KUKA KRL program: Bolge_1_Palet_Ort.src, Bolge_1_Palet_Ort.dat

--- Bolge_1_Palet_Ort.src ---
&ACCESS RVO1
&REL 27
&PARAM EDITMASK = *
&PARAM TEMPLATE = C:\KRC\Roboter\Template\vorgabe
&PARAM DISKPATH = KRC:\R1\Program\Sub_Rutinler
DEF Bolge_1_Palet_Ort( )
;FOLD INI;%{PE}
  ;FOLD BASISTECH INI
    GLOBAL INTERRUPT DECL 3 WHEN $STOPMESS==TRUE DO IR_STOPM ( )
    INTERRUPT ON 3
    BAS (#INITMOV,0 )
  ;ENDFOLD (BASISTECH INI)
  ;FOLD USER INI
    ;Make your modifications here

  ;ENDFOLD (USER INI)
;ENDFOLD (INI)

;;FOLD SPTP B1_Master Vel=100 % PDAT1 Tool[1]:Gripper Base[0] ;%{PE}
;;FOLD Parameters ;%{h}
;;Params IlfProvider=kukaroboter.basistech.inlineforms.movement.spline; Kuka.IsGlobalPoint=False; Kuka.PointName=B1_Master; Kuka.BlendingEnabled=False; Kuka.MoveDataPtpName=PDAT1; Kuka.VelocityPtp=100; Kuka.VelocityFieldEnabled=True; Kuka.ColDetectFieldEnabled=True; Kuka.CurrentCDSetIndex=0; Kuka.MovementParameterFieldEnabled=True; IlfCommand=SPTP
;;ENDFOLD
;SPTP XB1_Master WITH $VEL_AXIS[1] = SVEL_JOINT(100.0), $TOOL = STOOL2(FB1_Master), $BASE = SBASE(FB1_Master.BASE_NO), $IPO_MODE = SIPO_MODE(FB1_Master.IPO_FRAME), $LOAD = SLOAD(FB1_Master.TOOL_NO), $ACC_AXIS[1] = SACC_JOINT(PPDAT1), $APO = SAPO_PTP(PPDAT1), $GEAR_JERK[1] = SGEAR_JERK(PPDAT1), $COLLMON_TOL_PRO[1] = USE_CM_PRO_VALUES(0)
;;ENDFOLD

PaletMasterX=840
PaletMasterY=640

Base_Data[1]=Frame_Donustur(XB1_Master)
BASE_DATA[1].x=BASE_DATA[1].x-(PaletMasterX/2)
BASE_DATA[1].Y=BASE_DATA[1].Y-(PaletMasterY/2)

      IF (ParcaUzunluk<=1500)THEN

         BASE_DATA[1].x=BASE_DATA[1].x+(PaletUzunluk/2)
         BASE_DATA[1].Y=BASE_DATA[1].Y+(PaletGenislik/2)

      ENDIF

      IF (ParcaUzunluk>=1600) AND (ParcaUzunluk<=3000) THEN

         BASE_DATA[1].x=BASE_DATA[1].x+(PaletUzunluk/2)
         BASE_DATA[1].Y=BASE_DATA[1].Y+(PaletGenislik/2)

      ENDIF

END

DEFFCT FRAME Frame_Donustur(e6GeciciPos:IN)
   ;FOLD  Tanimlamalar
      DECL E6POS e6GeciciPos
      DECL FRAME ReturnFrame
   ;ENDFOLD
   ReturnFrame=$Nullframe
   ReturnFrame.X=e6GeciciPos.X
   ReturnFrame.Y=e6GeciciPos.Y
   ReturnFrame.Z=e6GeciciPos.Z
   ReturnFrame.A=e6GeciciPos.A
   ReturnFrame.B=e6GeciciPos.B
   ReturnFrame.C=e6GeciciPos.C
   RETURN ReturnFrame
ENDFCT

--- Bolge_1_Palet_Ort.dat ---
&ACCESS RVO1
&REL 25
&PARAM EDITMASK = *
&PARAM TEMPLATE = C:\KRC\Roboter\Template\vorgabe
&PARAM DISKPATH = KRC:\R1\Program\Sub_Rutinler
DEFDAT  BOLGE_1_PALET_ORT
;FOLD EXTERNAL DECLARATIONS;%{PE}%MKUKATPBASIS,%CEXT,%VCOMMON,%P
;FOLD BASISTECH EXT;%{PE}%MKUKATPBASIS,%CEXT,%VEXT,%P
EXT  BAS (BAS_COMMAND  :IN,REAL  :IN )
DECL INT SUCCESS
;ENDFOLD (BASISTECH EXT)
;FOLD USER EXT;%{E}%MKUKATPUSER,%CEXT,%VEXT,%P
;Make your modifications here

;ENDFOLD (USER EXT)
;ENDFOLD (EXTERNAL DECLARATIONS)
DECL E6POS XB1_Master={X 692.638489,Y 1644.84766,Z -1224.56201,A 0,B 0,C 0,S 6,T 19,E1 0.0,E2 0.0,E3 0.0,E4 0.0,E5 0.0,E6 0.0}
DECL FDAT FB1_Master={TOOL_NO 1,BASE_NO 0,IPO_FRAME #BASE,POINT2[] " "}
DECL PDAT PPDAT1={VEL 100.000,ACC 100.000,APO_DIST 500.000,APO_MODE #CDIS,GEAR_JERK 100.000,EXAX_IGN 0}
DECL MODULEPARAM_T LAST_TP_PARAMS={PARAMS[] "Kuka.VelocityFieldEnabled=False; Kuka.ColDetectFieldEnabled=False; Kuka.MovementParameterFieldEnabled=False; Kuka.IsAngleEnabled=False; Kuka.PointName=B1_Master; Kuka.FrameData.base_no=0; Kuka.FrameData.tool_no=1; Kuka.FrameData.ipo_frame=#BASE; Kuka.isglobalpoint=False; Kuka.MoveDataPtpName=PDAT1; Kuka.MovementDataPdat.apo_mode=#CDIS; Kuka.MovementDataPdat.apo_dist=500; Kuka.MovementData.vel=100; Kuka.MovementData.acc=100; Kuka.MovementData.exax_ign=0; Kuka.VelocityPtp=100; Kuka.BlendingEnabled=False; Kuka.APXEnabled=False; Kuka.CurrentCDSetIndex=0"}
DECL PDAT PPDAT2={VEL 100.000,ACC 100.000,APO_DIST 500.000,APO_MODE #CDIS,GEAR_JERK 100.000,EXAX_IGN 0}
DECL FDAT FB1_Master_1={TOOL_NO 1,BASE_NO 0,IPO_FRAME #BASE,POINT2[] " "}
DECL E6POS XB1_Master_1={X 2224.76123,Y -5.80455971,Z 416.847015,A 2.34930611,B -1.32013202E-13,C -3.04060856E-12,S 2,T 10,E1 0.0,E2 0.0,E3 0.0,E4 0.0,E5 0.0,E6 0.0}
ENDDAT
